KUKA KRL program: testcead.src, testcead.dat

--- testcead.src ---
&ACCESS RVO
&REL 87
&PARAM EDITMASK = *
&PARAM TEMPLATE = C:\KRC\Roboter\Template\vorgabe
&PARAM DISKPATH = KRC:\R1\Program\CNCR
DEF TestCEAD( )
DECL INT _i
;FOLD INI;%{PE}
  ;FOLD BASISTECH INI
    GLOBAL INTERRUPT DECL 3 WHEN $STOPMESS==TRUE DO IR_STOPM ( )
    INTERRUPT ON 3
GLOBAL INTERRUPT DECL 4 WHEN bCeadInterrupt== TRUE DO CeadInterrupt()
    INTERRUPT ON 4
    BAS (#INITMOV,0 )
  ;ENDFOLD (BASISTECH INI)
  ;FOLD USER INI
    ;Make your modifications here

  ;ENDFOLD (USER INI)
  ;ENDFOLD (INI)

;************************************************
;              CNC Robotics Ltd
;************************************************
;     Contact: helpdesk@cncrobotics.co.uk
;     Date: 26/09/23
;     Version: 0.18.51
;************************************************
; Description: Routine to test the cead extruder.
;************************************************

;BCO move so the program can be run in automatic
PTP $POS_ACT

;Clear cead errors is present
ResetCead()

;Set extruder perameters
rPumpTime = 30   ;Time(seconds) pump will pull material to the hopper
rShotSize = 1.0 ;Time(seconds) the pinch valve will open, allowing material through
SetPelletSource (#INTERNAL_CABINET) ;Set the source of material as the dryer
oBuzzOnEmpty = TRUE

;Set temperatures
SetHeatZones (160,170,180,180);

;Ready system
HeatersOn()
TransportOn()
WaitForReady()

;Start extrusion
SetScrewSpeed(10)
RotationOn()

;Allow extrusion to work so tests can be carried out
FOR _i= 1 TO 180
	WAIT SEC 3
   SetScrewSpeed(_i)
ENDFOR

;Change of heatzones while running should test over temp signals
SetHeatZones (230,240,250,250)

;Allow extrusion to work so tests can be carried out
FOR _i= 1 TO 180
	WAIT SEC 3
   SetScrewSpeed(_i)
ENDFOR

;Change of heatzones while running should test under temp signals
SetHeatZones (160,170,180,180);

;Allow extrusion to work so tests can be carried out
FOR _i= 1 TO 180
	WAIT SEC 3
   SetScrewSpeed(_i)
ENDFOR

;Finish program and turn off extruder
SetScrewSpeed(0)
FinishPrint()


END

--- testcead.dat ---
&ACCESS RVP
&REL 56
&PARAM EDITMASK = *
&PARAM TEMPLATE = C:\KRC\Roboter\Template\vorgabe
&PARAM DISKPATH = KRC:\R1\Program\CNCR
DEFDAT  TestCEAD
;FOLD EXTERNAL DECLARATIONS;%{PE}%MKUKATPBASIS,%CEXT,%VCOMMON,%P
;FOLD BASISTECH EXT;%{PE}%MKUKATPBASIS,%CEXT,%VEXT,%P
EXT  BAS (BAS_COMMAND  :IN,REAL  :IN )
DECL INT SUCCESS
;ENDFOLD (BASISTECH EXT)
;FOLD USER EXT;%{E}%MKUKATPUSER,%CEXT,%VEXT,%P
;Make your modifications here

;ENDFOLD (USER EXT)
;ENDFOLD (EXTERNAL DECLARATIONS)
DECL BASIS_SUGG_T LAST_BASIS={POINT1[] "P0                      ",POINT2[] "P0                      ",CP_PARAMS[] "CPDAT0                  ",PTP_PARAMS[] "PDAT0                   ",CONT[] "                        ",CP_VEL[] "2.0                     ",PTP_VEL[] "100                     ",SYNC_PARAMS[] "SYNCDAT                 ",SPL_NAME[] "S0                      ",A_PARAMS[] "ADAT0                   "}
DECL E6POS XP1={X 1044.07520,Y -1448.90295,Z 2604.21387,A -0.207003787,B 32.7573776,C 0.167719990,S 22,T 27,E1 1450.01270,E2 0.0,E3 0.0,E4 0.0,E5 0.0,E6 0.0}
DECL FDAT FP1={TOOL_NO 0,BASE_NO 0,IPO_FRAME #BASE,POINT2[] " "}
DECL PDAT PPDAT1={VEL 20.0000,ACC 100.000,APO_DIST 500.000,APO_MODE #CDIS,GEAR_JERK 100.000,EXAX_IGN 0}
DECL MODULEPARAM_T LAST_TP_PARAMS={PARAMS[] "Kuka.PointName=P1; Kuka.FrameData.base_no=0; Kuka.FrameData.tool_no=0; Kuka.FrameData.ipo_frame=#BASE; Kuka.isglobalpoint=False; Kuka.MoveDataPtpName=PDAT1; Kuka.MovementDataPdat.apo_mode=#CDIS; Kuka.MovementDataPdat.apo_dist=500; Kuka.MovementData.vel=20; Kuka.MovementData.acc=100; Kuka.MovementData.exax_ign=0; Kuka.VelocityPtp=20; Kuka.BlendingEnabled=False; Kuka.CurrentCDSetIndex=0           "}
DECL PDAT PPDAT2={VEL 20.0000,ACC 100.000,APO_DIST 500.000,APO_MODE #CDIS,GEAR_JERK 100.000,EXAX_IGN 0}
ENDDAT
